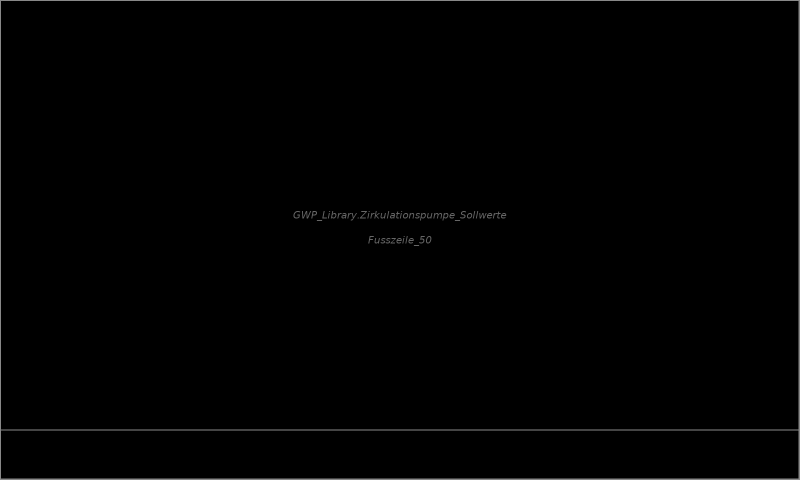
VISUALIZATION Zirkulationspumpe_Sollwerte  // 800x480
    Frame (0,0 800x430)
        shows GWP_Library.Zirkulationspumpe_Sollwerte(FB_Zirk_Pumpe := Main.Zirk_Pumpe_0)
    Frame (0,0 800x480)
        shows Fusszeile_50()
END_VISUALIZATION

(* stored: Version 1.1.0.1, ProductVersion 3.1.4022.6
   Visu Zirkulationspumpe_Sollwerte: Id {bd0f92b0-6353-49fa-9e0c-06cbc8f708fc} *)
